INTERFACE I_ForwardEnumerator EXTENDS I_Disposable

PROPERTY PUBLIC IsValid : BOOL
GET
END_GET
END_PROPERTY

METHOD PUBLIC MoveNext : BOOL
END_METHOD

METHOD Reset
VAR_INPUT
END_VAR
END_METHOD

METHOD PUBLIC TryGet : BOOL;
VAR_INPUT
    Destination : ANY;
END_VAR
END_METHOD

METHOD PUBLIC TryGetTo : BOOL;
VAR_INPUT
    DestinationAddress : PVOID;
    DestinationSize : UDINT;
END_VAR
END_METHOD

END_INTERFACE

(* stored: Version 1.1.0.1, ProductVersion 3.1.4024.12
   Itf I_ForwardEnumerator: Id {c34fbdaf-85cc-079c-2727-3c703d7faf71}
   Property IsValid: Id {e0014986-3f89-0842-16c5-0daf4dbae224}
   Get Get: Id {8c7b57be-c122-0e01-134a-a1b9a989a029}
   Method MoveNext: Id {b85a318f-280b-0b33-3a1b-2fd84090d5e4}
   Method Reset: Id {0f78e995-65f0-4ba9-9964-ba2117aa49e8}
   Method TryGet: Id {74e7636e-1bf0-072e-1443-81e758afc41b}
   Method TryGetTo: Id {27f1142b-c93b-09f4-098e-5eaf2edb7678} *)
